Fanuc KAREL source: kc00005.KL

-- PROVISIONAL review KL for V1013-1; original PC SHA256 c61e7d48ca0a923dcf5123ff44c66eee0f3d20326dfc0188aff4018340f30978
-- Incomplete behavior may be omitted. Consult companion uncertainty JSON. Do not deploy.
PROGRAM KC00005
%NOLOCKGROUP
BEGIN
  -- UNRESOLVED_PC offsets 5-27; opcodes 27,22,22,22,31
  -- UNRESOLVED_PC offsets 32-36; opcodes 7F
END KC00005
